// TIA Portal V18 export
FUNCTION "RTG1_POST" : Void   // FC17, LAD
{ S7_Optimized_Access := 'TRUE' }
// stored: SetENOAutomatically false
BEGIN

REGION Network 1: Send the acknowledgment telegram to RTG2
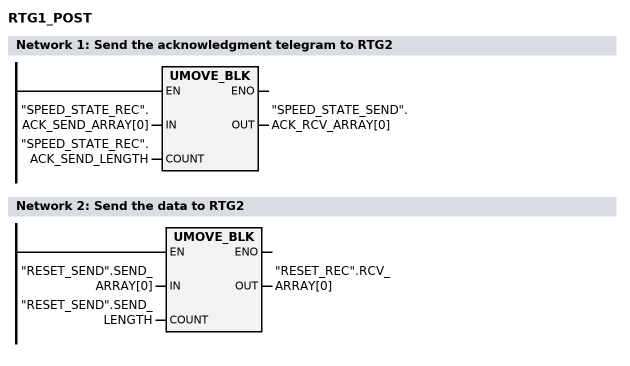
   UMOVE_BLK(IN := "SPEED_STATE_REC".ACK_SEND_ARRAY[0],
             COUNT := "SPEED_STATE_REC".ACK_SEND_LENGTH,
             OUT => "SPEED_STATE_SEND".ACK_RCV_ARRAY[0]);
END_REGION

REGION Network 2: Send the data to RTG2
   UMOVE_BLK(IN := "RESET_SEND".SEND_ARRAY[0],
             COUNT := "RESET_SEND".SEND_LENGTH,
             OUT => "RESET_REC".RCV_ARRAY[0]);
END_REGION
END_FUNCTION
